FUNCTION_BLOCK FB_TaskRunner_Test EXTENDS TcUnit.FB_TestSuite
VAR
END_VAR

_01_TrueIsTrue();

METHOD PRIVATE _01_TrueIsTrue
VAR
END_VAR
TEST('_01_TrueIsTrue');

AssertTrue(
	Condition := TRUE,
	Message := 'True should always be true'
);

TEST_FINISHED();
END_METHOD

END_FUNCTION_BLOCK

(* stored: Version 1.1.0.1, ProductVersion 3.1.4024.15
   POU FB_TaskRunner_Test: Id {d3f43d38-44f6-4522-94b7-30859937d93c}, SpecialFunc None
   Method _01_TrueIsTrue: Id {6358bad8-d4a6-48f3-9345-71976b3725f0} *)
